// TIA Portal project "FactoryIO_Template_S7-1200_V15" (V15)
// Vorlageprojekt für das Buch mit Zielsystem S7-1200

(* hardware
DEVICE "S7-1200-Station_1"  S7-1200 Station
   slot 0: "Baugruppenträger_0"  Rack  V1.0
   slot 1: "PLC_1"  CPU 1211C DC/DC/DC  6ES7 211-1AE40-0XB0  V4.1
*)

// ===== PLC "PLC_1"  CPU 1211C DC/DC/DC =====

VAR_GLOBAL   // PLC tag table "Standard-Variablentabelle"
   "Start" AT %E0.0 : Bool;
   "sensor1" AT %E0.1 : Bool;
   "sensor2" AT %I0.2 : Bool;
   "Conv1" AT %Q0.0 : Bool;
   "Conv2" AT %Q0.1 : Bool;
   "Tag_1" AT %M0.1 : Bool;
   "Tag_2" AT %M0.2 : Bool;
   "Tag_3" AT %M0.0 : Bool;
   "Counter_on" AT %Q0.2 : Bool;
   "Tag_5" AT %Q0.3 : Bool;
   "Tag_6" AT %M0.3 : Bool;
   "Tag_7" AT %M0.4 : Bool;
   "Tag_8" AT %I0.3 : Bool;
   "Tag_9" AT %M0.5 : Bool;
   "Tag_10" AT %M1.0 : Bool;
END_VAR

// folder: System blocks/Program resources

DATA_BLOCK "IEC_Counter_0_DB"   // DB1
{ S7_Optimized_Access := 'TRUE' }
AUTHOR : Simatic
FAMILY : IEC
NAME : CNTR
VERSION : 1.0
// stored: InstanceOfName IEC_COUNTER
"IEC_COUNTER"
BEGIN
END_DATA_BLOCK

// folder: (top level)

FUNCTION "MHJ-PLC-Lab-Function-S71200" : Void   // FC9000, SCL
{ S7_Optimized_Access := 'TRUE' }
VERSION : 0.1
   VAR_TEMP
      rdTimeReturn : Int;
      outputTime : DTL;
      SyncVal : Byte;
      forVal : Int;
      forVal_2 : Int;
      Value : Byte;
   END_VAR
   VAR CONSTANT
      CompVal : Byte := 16#34;
      Value_01 : Byte := 16#11;
      Value_01_DW : DWord := 16#A165_D992;
      Value_02_DW : DWord := 16#58BE_4401;
   END_VAR
BEGIN

   #Value:=PEEK(area := 16#82,
        dbNumber := 0,
        byteOffset := 511);
   #Value := #Value + 1;

   POKE(area := 16#82,
        dbNumber := 0,
        byteOffset := 511,
        value := #Value);

   POKE(area:=16#81,
        dbNumber:=0,
        byteOffset:=1016,
        value:=#Value_01_DW);
   POKE(area := 16#81,
        dbNumber := 0,
        byteOffset := 1020,
        value := #Value_02_DW);

   POKE(area := 16#81,
        dbNumber := 0,
        byteOffset := 511,
        value := B#16#00);

   FOR #forVal := 0 TO 120 DO
       FOR #forVal_2:=0 TO 10 DO
           #rdTimeReturn:=RD_SYS_T(#outputTime);
           #rdTimeReturn := WR_SYS_T(#outputTime);
           #rdTimeReturn := RD_SYS_T(#outputTime);
           #rdTimeReturn := WR_SYS_T(#outputTime);
       END_FOR;
       #SyncVal:= PEEK(area := 16#81,
                      dbNumber := 0,
                      byteOffset := 511);
       IF #SyncVal = #CompVal THEN
          GOTO M_1;
       END_IF;
   END_FOR;
   RETURN;

   M_1:
   POKE(area := 16#81,
        dbNumber := 0,
        byteOffset := 511,
        value := B#16#0);
END_FUNCTION

ORGANIZATION_BLOCK "Main"   // OB1, LAD, ProgramCycle
TITLE = "Main Program Sweep (Cycle)"
{ S7_Optimized_Access := 'TRUE' }
VERSION : 0.1
   VAR_INPUT
      Initial_Call : Bool;   // Initial call of this OB
      Remanence : Bool;   // =True, if remanent data are available
   END_VAR
   VAR_TEMP   // added for the SCL form of the ladder/FBD networks
      _w1 : Bool;
      _w2 : Bool;
      _w3 : Bool;
      _w4 : Bool;
      _w5 : Bool;
   END_VAR
BEGIN

REGION Network 1: Konnektierungsbaustein für PLC-Lab
   // Im Netzwerk 1 wird der Konnektierungsbaustein für PLC-Lab aufgerufen.
   // Dieser Aufruf darf nicht entfernt werden!
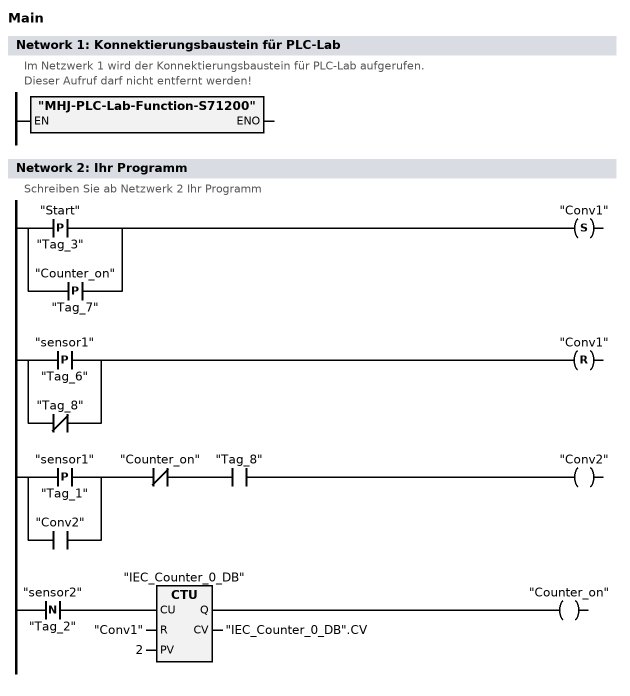
   RUNG wire#powerrail
      "MHJ-PLC-Lab-Function-S71200"()
   END_RUNG
   // the same network as SCL:
   "MHJ-PLC-Lab-Function-S71200"();
END_REGION

REGION Network 2: Ihr Programm
   // Schreiben Sie ab Netzwerk 2 Ihr Programm
   #_w1 := "Start" AND NOT "Tag_3";   // rising edge of "Start"
   "Tag_3" := "Start";
   #_w2 := "Counter_on" AND NOT "Tag_7";   // rising edge of "Counter_on"
   "Tag_7" := "Counter_on";
   IF #_w1 OR #_w2 THEN "Conv1" := TRUE; END_IF;
   #_w3 := "sensor1" AND NOT "Tag_6";   // rising edge of "sensor1"
   "Tag_6" := "sensor1";
   IF #_w3 OR NOT "Tag_8" THEN "Conv1" := FALSE; END_IF;
   #_w4 := "sensor1" AND NOT "Tag_1";   // rising edge of "sensor1"
   "Tag_1" := "sensor1";
   "Conv2" := (#_w4 OR "Conv2") AND NOT "Counter_on" AND "Tag_8";
   #_w5 := NOT "sensor2" AND "Tag_2";   // falling edge of "sensor2"
   "Tag_2" := "sensor2";
   "IEC_Counter_0_DB".CTU(CU := #_w5, R := "Conv1", PV := 2, CV => "IEC_Counter_0_DB".CV);
   "Counter_on" := "IEC_Counter_0_DB".Q;
END_REGION
END_ORGANIZATION_BLOCK